// TIA Portal V17 export
// export: Created 2023-02-14T02:49:06.1157461Z, ExportSetting WithDefaults, DisplayName Totally Integrated Automation Portal, DisplayVersion V17, DisplayName TIA Portal Openness, DisplayVersion V17, DisplayName TIA Portal Teamcenter Gateway, DisplayVersion V17, DisplayName TIA Portal Version Control Interface, DisplayVersion V17, DisplayName SINAMICS Startdrive Advanced, DisplayVersion V17, DisplayName SINAMICS Startdrive G130, G150, S120, S150, SINAMICS MV, S210, DisplayVersion V17, DisplayName SINAMICS Startdrive G110M, G120, G120C, G120D, G120P, G115D, DisplayVersion V17, DisplayName STEP 7 Professional, DisplayVersion V17, DisplayName STEP 7 Safety, DisplayVersion V17, DisplayName WinCC Professional, DisplayVersion V17
FUNCTION_BLOCK "DOSE"   // FB102, LAD
TITLE = Dosing Module type 1; 1 adustable speed pump and 1 auto valve.
{ S7_Optimized_Access := 'FALSE' }
AUTHOR : N@wi
FAMILY : DOSE
NAME : DOSE
VERSION : 0.1
// Dosing Module type 1:
// Use for Dosing module with adjustable speed pump and auto valve. Coarse dosing 
// and Fine dosing by adjusting the pump speed.
// stored: AutoNumber false, IsIECCheckEnabled false, SetENOAutomatically false, UDAEnableTagReadback false
   VAR_INPUT
      ISTART_COND : Bool;   // Starting Condition. 1 = Dose sequence can be Start
      IOP_COND : Bool;   // Operating Condition. 0 = Dose will be hold
      V_CLOSE : Bool;   // Valve in close position
      V_OPEN : Bool;   // Valve in open position
      P_RUN : Bool;   // Pump Run
      P_STOP : Bool;   // Pump Stop
      OP_MODE : Bool := TRUE;   // Dosing Mode; 0 = MANUAL; 1 = AUTO
      ISTART_AUT : Bool;   // Start command in Auto dosing mode
      IHOLD_AUT : Bool;   // Hold command in Auto dosing mode
      ISTOP_AUT : Bool;   // Stop command in Auto dosing mode
      ICOMP_AUT : Bool;   // Complete command in Auto dosing mode
      MON_EN : Bool;   // Monitoring time enable
      "Pulse 1HZ" : Bool;
      ACT_QTY : Real;   // Actual Counter quantity
      MON_TIME : Real := 60.0;   // Monitoring Time (in second)
      SP_DOSEQTY : Real;   // Dosing Setpoint Quantity
      SP_FINEQTY : Real;   // Fine Quantity Setpoint
      SP_IdleSPEED : Real;
      SP_FINESPEED : Real;   // Fine Speed Setpoint
      SP_COARSESPEED : Real;   // Coarse Speed Setpoint
      SAMPLE_T : Real := 1.0;   // Sample Time
      SETTLE_T : Real := 3.0;   // Settling Time
      INF_PERC : Real := 2.0;   // Percentage of calculated infligh qty (in %)
      LDT : Date_And_Time;
   END_VAR
   VAR_OUTPUT
      QAUTO : Bool;   // Selected Operation Mode 0 = MANUAL; 1 = AUTO
      QIDLE : Bool;   // Dosing module in IDLE state
      QDOSERun : Bool;   // Dosing module in Running state
      QFinish : Bool;   // Dosing module in Finish
      QSTARTING : Bool;   // Dosing module in STARTING state
      QHOLDING : Bool;   // Dosing module in HOLDING state
      QHELD : Bool;   // Dosing module in HELD state
      QSTOPPING : Bool;   // Dosing module in STOPPING state
      QSTOPPED : Bool;   // Dosing module in STOPPED state
      QSTART_COND : Bool;   // Starting Condition are met
      QOP_COND : Bool;   // Operating Condition are met
      QERR : Bool;   // General Error
      QERR_MON : Bool;   // Error cause by runtime monitoring error
      QERR_OP : Bool;   // Error cause by operating condition not OK
      QERR_START : Bool;   // Error cause by start condition not OK
      P_CMD : Bool;   // Pump Start command
      V_CMD : Bool;   // Valve Open command
      COUNT_RESET : Bool;   // Counter reset command
      QDoseComplete : Bool;
      P_SPEED : Real;   // Pump speed setpoint
      DOSED_QTY : Real;   // Dosed quantity
      ACT_MON_TIME : Real;   // Actual Monitoring Time
      Dose_State : Word;
   END_VAR
   VAR_IN_OUT
      IQOPSTART : Bool;   // Start command by operator in Manual dosing mode
      IQOPHOLD : Bool;   // Hold command by operator in Manual dosing mode
      IQOPSTOP : Bool;   // Stop command by operator in Manual dosing mode
      IQOPCOMPLETE : Bool;   // Complete command by operator in Manual dosing mode
      IQRESET : Bool;   // Reset Error
      IQINFL_QTY : Real := 3.0e+0;   // Inflight quantity. Will be calculated in end of dosing for the next dosing.
      IQSTEP : Int;   // Actual step
      IQRB_STEP : Int;   // Roll Back Step
   END_VAR
   VAR DB_SPECIFIC
      b_IDLE : Bool;   // Dosing module in IDLE state
      b_Finish : Bool;   // Dosing module in Finish state
      b_STARTING : Bool;   // Dosing module in STARTING state
      b_HOLDING : Bool;   // Dosing module in HOLDING state
      b_HELD : Bool;   // Dosing module in HELD state
      b_STOPPING : Bool;   // Dosing module in STOPPING state
      b_STOPPED : Bool;   // Dosing module in STOPPED state
      b_START : Bool;   // Start command
      b_HOLD : Bool;   // Hold command
      b_STOP : Bool;   // Stop command
      b_COMP : Bool;   // Complete command
      b_START_AP : Bool;   // Start command Auto Pulse
      b_HOLD_AP : Bool;   // Hold command Auto Pulse
      b_STOP_AP : Bool;   // Stop command Auto Pulse
      b_COMP_AP : Bool;   // Complete command Auto Pulse
      b_START_MP : Bool;   // Start command Manual Pulse
      b_HOLD_MP : Bool;   // Hold command Manual Pulse
      b_STOP_MP : Bool;   // Stop command Manual Pulse
      b_COMP_MP : Bool;   // Complete command Manual Pulse
      b_ERR_MON : Bool;   // Error cause by runtime monitoring error
      b_ERR_OP : Bool;   // Error cause by operating condition not OK
      b_ERR_START : Bool;   // Error cause by start condition not OK
      PE_Setle : Bool;
      PE_Mon : Bool;
      CMD_STEP : Int;   // STEP command
      r_MON : Real;   // Actual Monitoring Time
      r_STOP : Real;   // Quantity to stop dosing
      r_FINE : Real;   // Quantity change to fine dosing
      r_SETTLE_T : Real;   // Settling Time
      r_INFLIGHT : Real;   // Saved inflight qty
      r_DIFF : Real;   // Dosed Qty - SP Quantity
      r_INFDIFF : Real;   // Diff of Inflight qty to be added to new inflight
      r_INFPERC { ExternalAccessible := 'False'; ExternalVisible := 'False'; ExternalWritable := 'False'} : Real;
      LDT_Start { S7_SetPoint := 'True'} : Date_And_Time;
      LDT_Finish : Date_And_Time;
      TimeDose : Time;
      LastTimeDose : Time;
      PE_LDTStart : Bool;
      PE_LDTFinish : Bool;
      PE_LDTStore : Bool;
      PE_QtyStart : Bool;
      PE_QtyFinish : Bool;
      PE_QtyStore : Bool;
      AlwaysON : Bool;
      LastQtyDose : Real;
   END_VAR
   VAR_TEMP   // added for the SCL form of the ladder/FBD networks
      _w1 : Bool;
      _w2 : Bool;
      _w3 : Bool;
      _w4 : Bool;
   END_VAR
BEGIN

REGION Network 1: AlwaysON
   // Copying the command step number to actual step number to avoid double step in 
   // one scan.
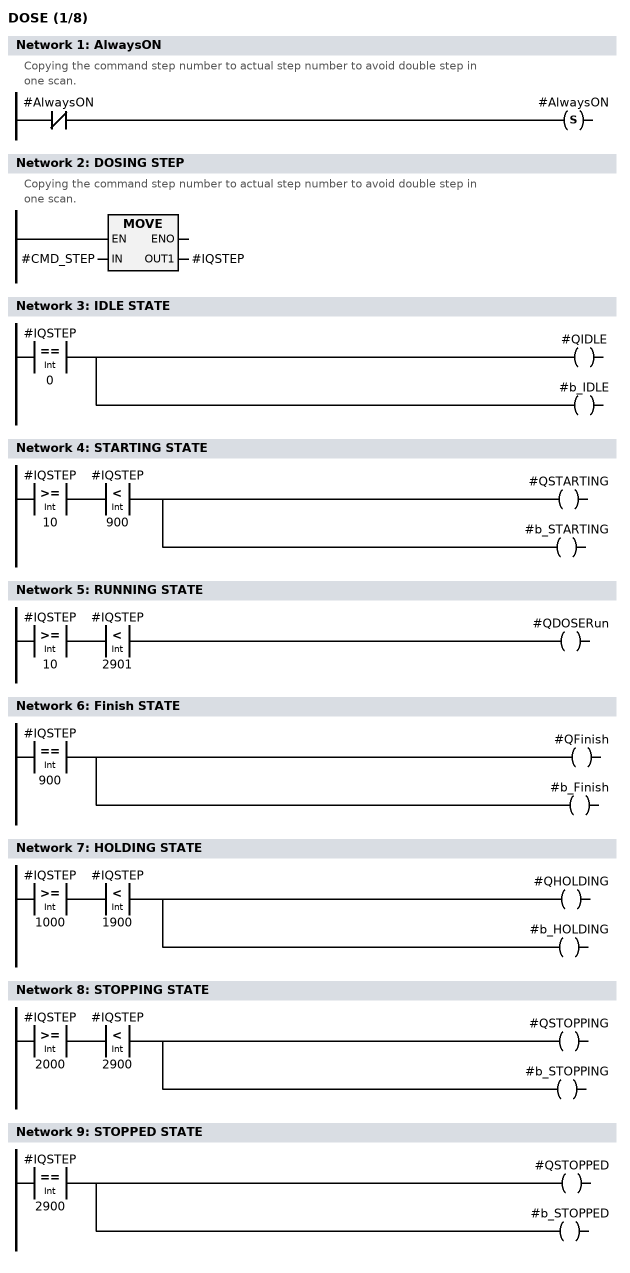
   RUNG wire#powerrail
      I_Contact( #AlwaysON )
      S_Coil( #AlwaysON )
   END_RUNG
   // the same network as SCL:
   IF NOT #AlwaysON THEN #AlwaysON := TRUE; END_IF;
END_REGION

REGION Network 2: DOSING STEP
   // Copying the command step number to actual step number to avoid double step in 
   // one scan.
   RUNG wire#powerrail
      { S7_GenerateENO := "TRUE" } Move(in := #CMD_STEP, out1 => #IQSTEP)
   END_RUNG
   // the same network as SCL:
   #IQSTEP := #CMD_STEP;
END_REGION

REGION Network 3: IDLE STATE
   RUNG wire#powerrail
      { S7_Templates := "SrcType := Int" } EQ_Contact(in1 := #IQSTEP, in2 := 0)
      wire#w1
      Coil( #QIDLE )
   END_RUNG
   RUNG wire#w1
      Coil( #b_IDLE )
   END_RUNG
   // the same network as SCL:
   #QIDLE := #IQSTEP = 0;
   #b_IDLE := #QIDLE;
END_REGION

REGION Network 4: STARTING STATE
   RUNG wire#powerrail
      { S7_Templates := "SrcType := Int" } GE_Contact(in1 := #IQSTEP, in2 := 10)
      { S7_Templates := "SrcType := Int" } LT_Contact(in1 := #IQSTEP, in2 := 900)
      wire#w1
      Coil( #QSTARTING )
   END_RUNG
   RUNG wire#w1
      Coil( #b_STARTING )
   END_RUNG
   // the same network as SCL:
   #QSTARTING := (#IQSTEP >= 10) AND (#IQSTEP < 900);
   #b_STARTING := #QSTARTING;
END_REGION

REGION Network 5: RUNNING STATE
   RUNG wire#powerrail
      { S7_Templates := "SrcType := Int" } GE_Contact(in1 := #IQSTEP, in2 := 10)
      { S7_Templates := "SrcType := Int" } LT_Contact(in1 := #IQSTEP, in2 := 2901)
      Coil( #QDOSERun )
   END_RUNG
   // the same network as SCL:
   #QDOSERun := (#IQSTEP >= 10) AND (#IQSTEP < 2901);
END_REGION

REGION Network 6: Finish STATE
   RUNG wire#powerrail
      { S7_Templates := "SrcType := Int" } EQ_Contact(in1 := #IQSTEP, in2 := 900)
      wire#w1
      Coil( #QFinish )
   END_RUNG
   RUNG wire#w1
      Coil( #b_Finish )
   END_RUNG
   // the same network as SCL:
   #QFinish := #IQSTEP = 900;
   #b_Finish := #QFinish;
END_REGION

REGION Network 7: HOLDING STATE
   RUNG wire#powerrail
      { S7_Templates := "SrcType := Int" } GE_Contact(in1 := #IQSTEP, in2 := 1000)
      { S7_Templates := "SrcType := Int" } LT_Contact(in1 := #IQSTEP, in2 := 1900)
      wire#w1
      Coil( #QHOLDING )
   END_RUNG
   RUNG wire#w1
      Coil( #b_HOLDING )
   END_RUNG
   // the same network as SCL:
   #QHOLDING := (#IQSTEP >= 1000) AND (#IQSTEP < 1900);
   #b_HOLDING := #QHOLDING;
END_REGION

REGION Network 8: STOPPING STATE
   RUNG wire#powerrail
      { S7_Templates := "SrcType := Int" } GE_Contact(in1 := #IQSTEP, in2 := 2000)
      { S7_Templates := "SrcType := Int" } LT_Contact(in1 := #IQSTEP, in2 := 2900)
      wire#w1
      Coil( #QSTOPPING )
   END_RUNG
   RUNG wire#w1
      Coil( #b_STOPPING )
   END_RUNG
   // the same network as SCL:
   #QSTOPPING := (#IQSTEP >= 2000) AND (#IQSTEP < 2900);
   #b_STOPPING := #QSTOPPING;
END_REGION

REGION Network 9: STOPPED STATE
   RUNG wire#powerrail
      { S7_Templates := "SrcType := Int" } EQ_Contact(in1 := #IQSTEP, in2 := 2900)
      wire#w1
      Coil( #QSTOPPED )
   END_RUNG
   RUNG wire#w1
      Coil( #b_STOPPED )
   END_RUNG
   // the same network as SCL:
   #QSTOPPED := #IQSTEP = 2900;
   #b_STOPPED := #QSTOPPED;
END_REGION

REGION Network 10: START COMMAND
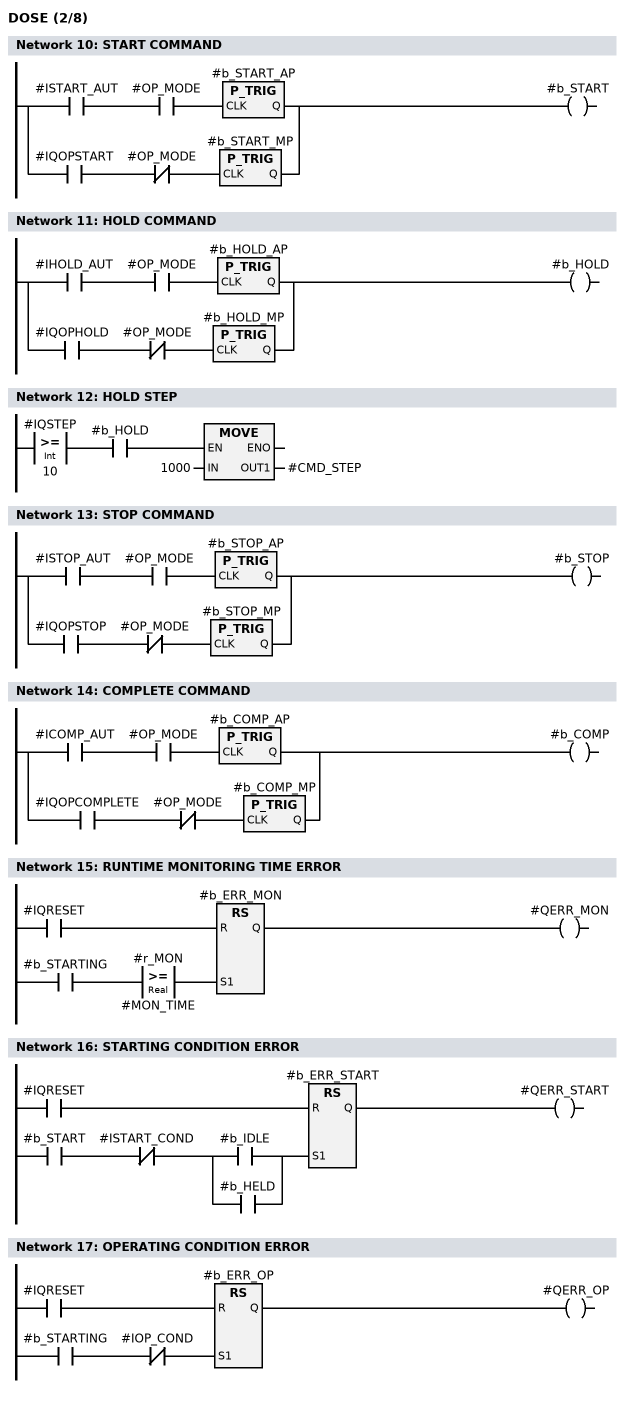
   RUNG wire#powerrail
      Contact( #ISTART_AUT )
      Contact( #OP_MODE )
      P_Trig( #b_START_AP )
      wire#w1
      Coil( #b_START )
   END_RUNG
   RUNG wire#powerrail
      Contact( #IQOPSTART )
      I_Contact( #OP_MODE )
      P_Trig( #b_START_MP )
   END_RUNG wire#w1
   // the same network as SCL:
   #_w1 := #ISTART_AUT AND #OP_MODE;
   #_w2 := #_w1 AND NOT #b_START_AP;   // rising edge
   #b_START_AP := #_w1;
   #_w3 := #IQOPSTART AND NOT #OP_MODE;
   #_w4 := #_w3 AND NOT #b_START_MP;   // rising edge
   #b_START_MP := #_w3;
   #b_START := #_w2 OR #_w4;
END_REGION

REGION Network 11: HOLD COMMAND
   RUNG wire#powerrail
      Contact( #IHOLD_AUT )
      Contact( #OP_MODE )
      P_Trig( #b_HOLD_AP )
      wire#w1
      Coil( #b_HOLD )
   END_RUNG
   RUNG wire#powerrail
      Contact( #IQOPHOLD )
      I_Contact( #OP_MODE )
      P_Trig( #b_HOLD_MP )
   END_RUNG wire#w1
   // the same network as SCL:
   #_w1 := #IHOLD_AUT AND #OP_MODE;
   #_w2 := #_w1 AND NOT #b_HOLD_AP;   // rising edge
   #b_HOLD_AP := #_w1;
   #_w3 := #IQOPHOLD AND NOT #OP_MODE;
   #_w4 := #_w3 AND NOT #b_HOLD_MP;   // rising edge
   #b_HOLD_MP := #_w3;
   #b_HOLD := #_w2 OR #_w4;
END_REGION

REGION Network 12: HOLD STEP
   RUNG wire#powerrail
      { S7_Templates := "SrcType := Int" } GE_Contact(in1 := #IQSTEP, in2 := 10)
      Contact( #b_HOLD )
      { S7_GenerateENO := "TRUE" } Move(in := 1000, out1 => #CMD_STEP)
   END_RUNG
   // the same network as SCL:
   IF (#IQSTEP >= 10) AND #b_HOLD THEN #CMD_STEP := 1000; END_IF;
END_REGION

REGION Network 13: STOP COMMAND
   RUNG wire#powerrail
      Contact( #ISTOP_AUT )
      Contact( #OP_MODE )
      P_Trig( #b_STOP_AP )
      wire#w1
      Coil( #b_STOP )
   END_RUNG
   RUNG wire#powerrail
      Contact( #IQOPSTOP )
      I_Contact( #OP_MODE )
      P_Trig( #b_STOP_MP )
   END_RUNG wire#w1
   // the same network as SCL:
   #_w1 := #ISTOP_AUT AND #OP_MODE;
   #_w2 := #_w1 AND NOT #b_STOP_AP;   // rising edge
   #b_STOP_AP := #_w1;
   #_w3 := #IQOPSTOP AND NOT #OP_MODE;
   #_w4 := #_w3 AND NOT #b_STOP_MP;   // rising edge
   #b_STOP_MP := #_w3;
   #b_STOP := #_w2 OR #_w4;
END_REGION

REGION Network 14: COMPLETE COMMAND
   RUNG wire#powerrail
      Contact( #ICOMP_AUT )
      Contact( #OP_MODE )
      P_Trig( #b_COMP_AP )
      wire#w1
      Coil( #b_COMP )
   END_RUNG
   RUNG wire#powerrail
      Contact( #IQOPCOMPLETE )
      I_Contact( #OP_MODE )
      P_Trig( #b_COMP_MP )
   END_RUNG wire#w1
   // the same network as SCL:
   #_w1 := #ICOMP_AUT AND #OP_MODE;
   #_w2 := #_w1 AND NOT #b_COMP_AP;   // rising edge
   #b_COMP_AP := #_w1;
   #_w3 := #IQOPCOMPLETE AND NOT #OP_MODE;
   #_w4 := #_w3 AND NOT #b_COMP_MP;   // rising edge
   #b_COMP_MP := #_w3;
   #b_COMP := #_w2 OR #_w4;
END_REGION

REGION Network 15: RUNTIME MONITORING TIME ERROR
   RUNG wire#powerrail
      Contact( #IQRESET )
      S_RS(operand := #b_ERR_MON, s1 := wire#w1)
      Coil( #QERR_MON )
   END_RUNG
   RUNG wire#powerrail
      Contact( #b_STARTING )
      { S7_Templates := "SrcType := Real" } GE_Contact(in1 := #r_MON, in2 := #MON_TIME)
   END_RUNG wire#w1
   // the same network as SCL:
   IF #IQRESET THEN
       #b_ERR_MON := FALSE;   // RS flip-flop
   END_IF;
   IF #b_STARTING AND (#r_MON >= #MON_TIME) THEN #b_ERR_MON := TRUE; END_IF;
   #QERR_MON := #b_ERR_MON;
END_REGION

REGION Network 16: STARTING CONDITION ERROR
   RUNG wire#powerrail
      Contact( #IQRESET )
      S_RS(operand := #b_ERR_START, s1 := wire#w2)
      Coil( #QERR_START )
   END_RUNG
   RUNG wire#powerrail
      Contact( #b_START )
      I_Contact( #ISTART_COND )
      wire#w1
      Contact( #b_IDLE )
   END_RUNG wire#w2
   RUNG wire#w1
      Contact( #b_HELD )
   END_RUNG wire#w2
   // the same network as SCL:
   IF #IQRESET THEN
       #b_ERR_START := FALSE;   // RS flip-flop
   END_IF;
   IF #b_START AND NOT #ISTART_COND AND (#b_IDLE OR #b_HELD) THEN #b_ERR_START := TRUE; END_IF;
   #QERR_START := #b_ERR_START;
END_REGION

REGION Network 17: OPERATING CONDITION ERROR
   RUNG wire#powerrail
      Contact( #IQRESET )
      S_RS(operand := #b_ERR_OP, s1 := wire#w1)
      Coil( #QERR_OP )
   END_RUNG
   RUNG wire#powerrail
      Contact( #b_STARTING )
      I_Contact( #IOP_COND )
   END_RUNG wire#w1
   // the same network as SCL:
   IF #IQRESET THEN
       #b_ERR_OP := FALSE;   // RS flip-flop
   END_IF;
   IF #b_STARTING AND NOT #IOP_COND THEN #b_ERR_OP := TRUE; END_IF;
   #QERR_OP := #b_ERR_OP;
END_REGION

REGION Network 18: GENERAL ERROR
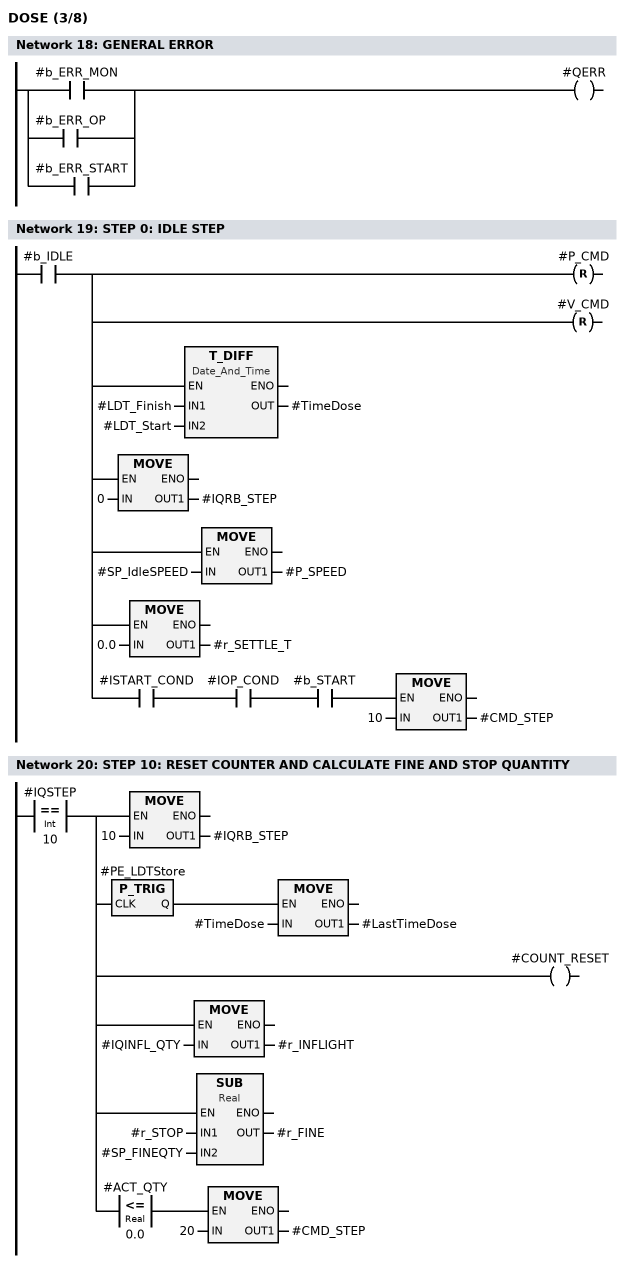
   RUNG wire#powerrail
      Contact( #b_ERR_MON )
      wire#w1
      Coil( #QERR )
   END_RUNG
   RUNG wire#powerrail
      Contact( #b_ERR_OP )
   END_RUNG wire#w1
   RUNG wire#powerrail
      Contact( #b_ERR_START )
   END_RUNG wire#w1
   // the same network as SCL:
   #QERR := #b_ERR_MON OR #b_ERR_OP OR #b_ERR_START;
END_REGION

REGION Network 19: STEP 0: IDLE STEP
   RUNG wire#powerrail
      Contact( #b_IDLE )
      wire#w1
      R_Coil( #P_CMD )
   END_RUNG
   RUNG wire#w1
      R_Coil( #V_CMD )
   END_RUNG
   RUNG wire#w1
      { S7_Templates := "[date_type := Date_And_Time, time_type := Time]" } T_DIFF(IN1 := #LDT_Finish, IN2 := #LDT_Start, OUT => #TimeDose)
   END_RUNG
   RUNG wire#w1
      { S7_GenerateENO := "TRUE" } Move(in := 0, out1 => #IQRB_STEP)
   END_RUNG
   RUNG wire#w1
      { S7_GenerateENO := "TRUE" } Move(in := #SP_IdleSPEED, out1 => #P_SPEED)
   END_RUNG
   RUNG wire#w1
      { S7_GenerateENO := "TRUE" } Move(in := 0.0, out1 => #r_SETTLE_T)
   END_RUNG
   RUNG wire#w1
      Contact( #ISTART_COND )
      Contact( #IOP_COND )
      Contact( #b_START )
      { S7_GenerateENO := "TRUE" } Move(in := 10, out1 => #CMD_STEP)
   END_RUNG
   // the same network as SCL:
   IF #b_IDLE THEN
       #P_CMD := FALSE;
       #V_CMD := FALSE;
       T_DIFF(IN1 := #LDT_Finish, IN2 := #LDT_Start, OUT => #TimeDose);
       #IQRB_STEP := 0;
       #P_SPEED := #SP_IdleSPEED;
       #r_SETTLE_T := 0.0;
   END_IF;
   IF #b_IDLE AND #ISTART_COND AND #IOP_COND AND #b_START THEN #CMD_STEP := 10; END_IF;
END_REGION

REGION Network 20: STEP 10: RESET COUNTER AND CALCULATE FINE AND STOP QUANTITY
   RUNG wire#powerrail
      { S7_Templates := "SrcType := Int" } EQ_Contact(in1 := #IQSTEP, in2 := 10)
      wire#w1
      { S7_GenerateENO := "TRUE" } Move(in := 10, out1 => #IQRB_STEP)
   END_RUNG
   RUNG wire#w1
      P_Trig( #PE_LDTStore )
      Move(in := #TimeDose, out1 => #LastTimeDose)
   END_RUNG
   RUNG wire#w1
      Coil( #COUNT_RESET )
   END_RUNG
   RUNG wire#w1
      { S7_GenerateENO := "TRUE" } Move(in := #IQINFL_QTY, out1 => #r_INFLIGHT)
   END_RUNG
   RUNG wire#w1
      { S7_Templates := "SrcType := Real"; S7_GenerateENO := "TRUE" } Sub(in1 := #r_STOP, in2 := #SP_FINEQTY, out => #r_FINE)
   END_RUNG
   RUNG wire#w1
      { S7_Templates := "SrcType := Real" } LE_Contact(in1 := #ACT_QTY, in2 := 0.0)
      { S7_GenerateENO := "TRUE" } Move(in := 20, out1 => #CMD_STEP)
   END_RUNG
   // the same network as SCL:
   #_w1 := #IQSTEP = 10;
   IF #_w1 THEN #IQRB_STEP := 10; END_IF;
   #_w2 := #_w1 AND NOT #PE_LDTStore;   // rising edge
   #PE_LDTStore := #_w1;
   IF #_w2 THEN #LastTimeDose := #TimeDose; END_IF;
   #COUNT_RESET := #_w1;
   IF #_w1 THEN
       #r_INFLIGHT := #IQINFL_QTY;
       #r_FINE := #r_STOP - #SP_FINEQTY;
   END_IF;
   IF #_w1 AND (#ACT_QTY <= 0.0) THEN #CMD_STEP := 20; END_IF;
END_REGION

REGION Network 21: STEP 20: OPEN VALVE
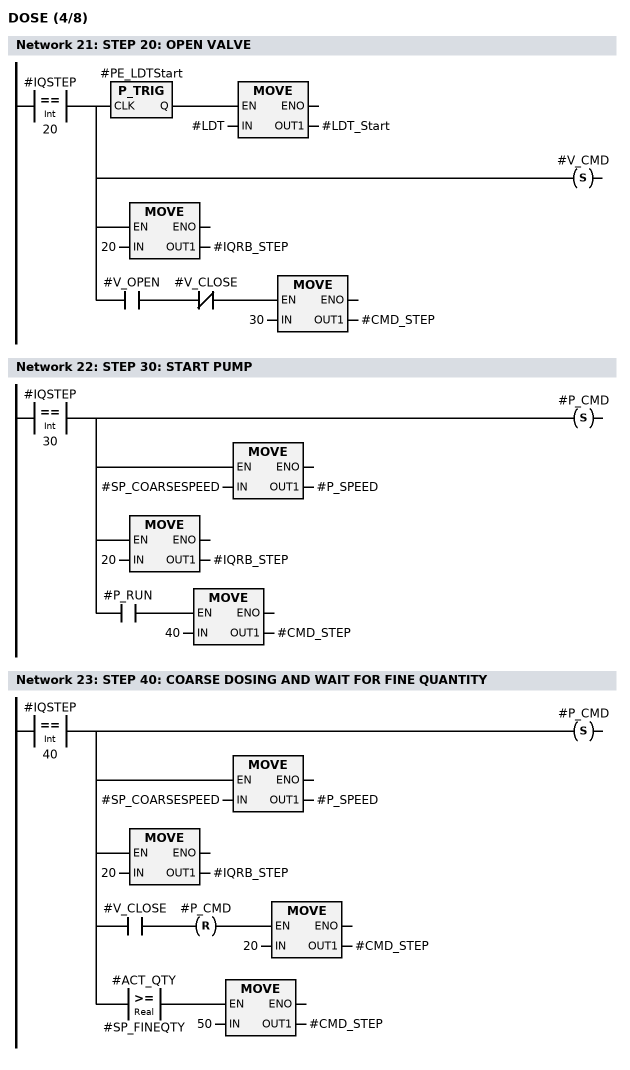
   RUNG wire#powerrail
      { S7_Templates := "SrcType := Int" } EQ_Contact(in1 := #IQSTEP, in2 := 20)
      wire#w1
      P_Trig( #PE_LDTStart )
      Move(in := #LDT, out1 => #LDT_Start)
   END_RUNG
   RUNG wire#w1
      S_Coil( #V_CMD )
   END_RUNG
   RUNG wire#w1
      { S7_GenerateENO := "TRUE" } Move(in := 20, out1 => #IQRB_STEP)
   END_RUNG
   RUNG wire#w1
      Contact( #V_OPEN )
      I_Contact( #V_CLOSE )
      { S7_GenerateENO := "TRUE" } Move(in := 30, out1 => #CMD_STEP)
   END_RUNG
   // the same network as SCL:
   #_w1 := #IQSTEP = 20;
   #_w2 := #_w1 AND NOT #PE_LDTStart;   // rising edge
   #PE_LDTStart := #_w1;
   IF #_w2 THEN #LDT_Start := #LDT; END_IF;
   IF #_w1 THEN
       #V_CMD := TRUE;
       #IQRB_STEP := 20;
   END_IF;
   IF #_w1 AND #V_OPEN AND NOT #V_CLOSE THEN #CMD_STEP := 30; END_IF;
END_REGION

REGION Network 22: STEP 30: START PUMP
   RUNG wire#powerrail
      { S7_Templates := "SrcType := Int" } EQ_Contact(in1 := #IQSTEP, in2 := 30)
      wire#w1
      S_Coil( #P_CMD )
   END_RUNG
   RUNG wire#w1
      { S7_GenerateENO := "TRUE" } Move(in := #SP_COARSESPEED, out1 => #P_SPEED)
   END_RUNG
   RUNG wire#w1
      { S7_GenerateENO := "TRUE" } Move(in := 20, out1 => #IQRB_STEP)
   END_RUNG
   RUNG wire#w1
      Contact( #P_RUN )
      { S7_GenerateENO := "TRUE" } Move(in := 40, out1 => #CMD_STEP)
   END_RUNG
   // the same network as SCL:
   #_w1 := #IQSTEP = 30;
   IF #_w1 THEN
       #P_CMD := TRUE;
       #P_SPEED := #SP_COARSESPEED;
       #IQRB_STEP := 20;
   END_IF;
   IF #_w1 AND #P_RUN THEN #CMD_STEP := 40; END_IF;
END_REGION

REGION Network 23: STEP 40: COARSE DOSING AND WAIT FOR FINE QUANTITY
   RUNG wire#powerrail
      { S7_Templates := "SrcType := Int" } EQ_Contact(in1 := #IQSTEP, in2 := 40)
      wire#w1
      S_Coil( #P_CMD )
   END_RUNG
   RUNG wire#w1
      { S7_GenerateENO := "TRUE" } Move(in := #SP_COARSESPEED, out1 => #P_SPEED)
   END_RUNG
   RUNG wire#w1
      { S7_GenerateENO := "TRUE" } Move(in := 20, out1 => #IQRB_STEP)
   END_RUNG
   RUNG wire#w1
      Contact( #V_CLOSE )
      R_Coil( #P_CMD )
      { S7_GenerateENO := "TRUE" } Move(in := 20, out1 => #CMD_STEP)
   END_RUNG
   RUNG wire#w1
      { S7_Templates := "SrcType := Real" } GE_Contact(in1 := #ACT_QTY, in2 := #SP_FINEQTY)
      { S7_GenerateENO := "TRUE" } Move(in := 50, out1 => #CMD_STEP)
   END_RUNG
   // the same network as SCL:
   #_w1 := #IQSTEP = 40;
   IF #_w1 THEN
       #P_CMD := TRUE;
       #P_SPEED := #SP_COARSESPEED;
       #IQRB_STEP := 20;
   END_IF;
   IF #_w1 AND #V_CLOSE THEN
       #P_CMD := FALSE;
       #CMD_STEP := 20;
   END_IF;
   IF #_w1 AND (#ACT_QTY >= #SP_FINEQTY) THEN #CMD_STEP := 50; END_IF;
END_REGION

REGION Network 24: STEP 50: FINE DOSING AND WAIT FOR STOP QUANTITY
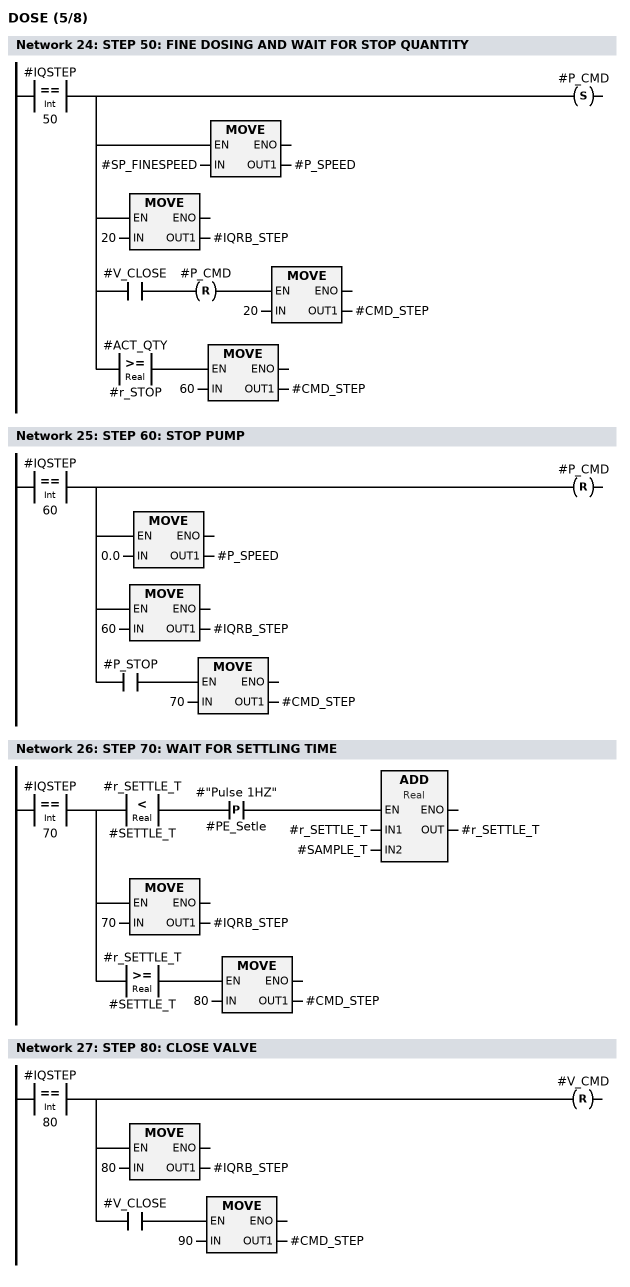
   RUNG wire#powerrail
      { S7_Templates := "SrcType := Int" } EQ_Contact(in1 := #IQSTEP, in2 := 50)
      wire#w1
      S_Coil( #P_CMD )
   END_RUNG
   RUNG wire#w1
      { S7_GenerateENO := "TRUE" } Move(in := #SP_FINESPEED, out1 => #P_SPEED)
   END_RUNG
   RUNG wire#w1
      { S7_GenerateENO := "TRUE" } Move(in := 20, out1 => #IQRB_STEP)
   END_RUNG
   RUNG wire#w1
      Contact( #V_CLOSE )
      R_Coil( #P_CMD )
      { S7_GenerateENO := "TRUE" } Move(in := 20, out1 => #CMD_STEP)
   END_RUNG
   RUNG wire#w1
      { S7_Templates := "SrcType := Real" } GE_Contact(in1 := #ACT_QTY, in2 := #r_STOP)
      { S7_GenerateENO := "TRUE" } Move(in := 60, out1 => #CMD_STEP)
   END_RUNG
   // the same network as SCL:
   #_w1 := #IQSTEP = 50;
   IF #_w1 THEN
       #P_CMD := TRUE;
       #P_SPEED := #SP_FINESPEED;
       #IQRB_STEP := 20;
   END_IF;
   IF #_w1 AND #V_CLOSE THEN
       #P_CMD := FALSE;
       #CMD_STEP := 20;
   END_IF;
   IF #_w1 AND (#ACT_QTY >= #r_STOP) THEN #CMD_STEP := 60; END_IF;
END_REGION

REGION Network 25: STEP 60: STOP PUMP
   RUNG wire#powerrail
      { S7_Templates := "SrcType := Int" } EQ_Contact(in1 := #IQSTEP, in2 := 60)
      wire#w1
      R_Coil( #P_CMD )
   END_RUNG
   RUNG wire#w1
      { S7_GenerateENO := "TRUE" } Move(in := 0.0, out1 => #P_SPEED)
   END_RUNG
   RUNG wire#w1
      { S7_GenerateENO := "TRUE" } Move(in := 60, out1 => #IQRB_STEP)
   END_RUNG
   RUNG wire#w1
      Contact( #P_STOP )
      { S7_GenerateENO := "TRUE" } Move(in := 70, out1 => #CMD_STEP)
   END_RUNG
   // the same network as SCL:
   #_w1 := #IQSTEP = 60;
   IF #_w1 THEN
       #P_CMD := FALSE;
       #P_SPEED := 0.0;
       #IQRB_STEP := 60;
   END_IF;
   IF #_w1 AND #P_STOP THEN #CMD_STEP := 70; END_IF;
END_REGION

REGION Network 26: STEP 70: WAIT FOR SETTLING TIME
   RUNG wire#powerrail
      { S7_Templates := "SrcType := Int" } EQ_Contact(in1 := #IQSTEP, in2 := 70)
      wire#w1
      { S7_Templates := "SrcType := Real" } LT_Contact(in1 := #r_SETTLE_T, in2 := #SETTLE_T)
      P_Contact(operand := #"Pulse 1HZ", bit := #PE_Setle)
      { S7_Templates := "SrcType := Real"; S7_GenerateENO := "TRUE" } Add(in1 := #r_SETTLE_T, in2 := #SAMPLE_T, out => #r_SETTLE_T)
   END_RUNG
   RUNG wire#w1
      { S7_GenerateENO := "TRUE" } Move(in := 70, out1 => #IQRB_STEP)
   END_RUNG
   RUNG wire#w1
      { S7_Templates := "SrcType := Real" } GE_Contact(in1 := #r_SETTLE_T, in2 := #SETTLE_T)
      { S7_GenerateENO := "TRUE" } Move(in := 80, out1 => #CMD_STEP)
   END_RUNG
   // the same network as SCL:
   #_w1 := #IQSTEP = 70;
   #_w2 := #_w1 AND (#r_SETTLE_T < #SETTLE_T) AND #"Pulse 1HZ" AND NOT #PE_Setle;   // rising edge of #"Pulse 1HZ"
   #PE_Setle := #"Pulse 1HZ";
   IF #_w2 THEN #r_SETTLE_T := #r_SETTLE_T + #SAMPLE_T; END_IF;
   IF #_w1 THEN #IQRB_STEP := 70; END_IF;
   IF #_w1 AND (#r_SETTLE_T >= #SETTLE_T) THEN #CMD_STEP := 80; END_IF;
END_REGION

REGION Network 27: STEP 80: CLOSE VALVE
   RUNG wire#powerrail
      { S7_Templates := "SrcType := Int" } EQ_Contact(in1 := #IQSTEP, in2 := 80)
      wire#w1
      R_Coil( #V_CMD )
   END_RUNG
   RUNG wire#w1
      { S7_GenerateENO := "TRUE" } Move(in := 80, out1 => #IQRB_STEP)
   END_RUNG
   RUNG wire#w1
      Contact( #V_CLOSE )
      { S7_GenerateENO := "TRUE" } Move(in := 90, out1 => #CMD_STEP)
   END_RUNG
   // the same network as SCL:
   #_w1 := #IQSTEP = 80;
   IF #_w1 THEN
       #V_CMD := FALSE;
       #IQRB_STEP := 80;
   END_IF;
   IF #_w1 AND #V_CLOSE THEN #CMD_STEP := 90; END_IF;
END_REGION

REGION Network 28: STEP 90: CALCULATE INFLIGHT QTY
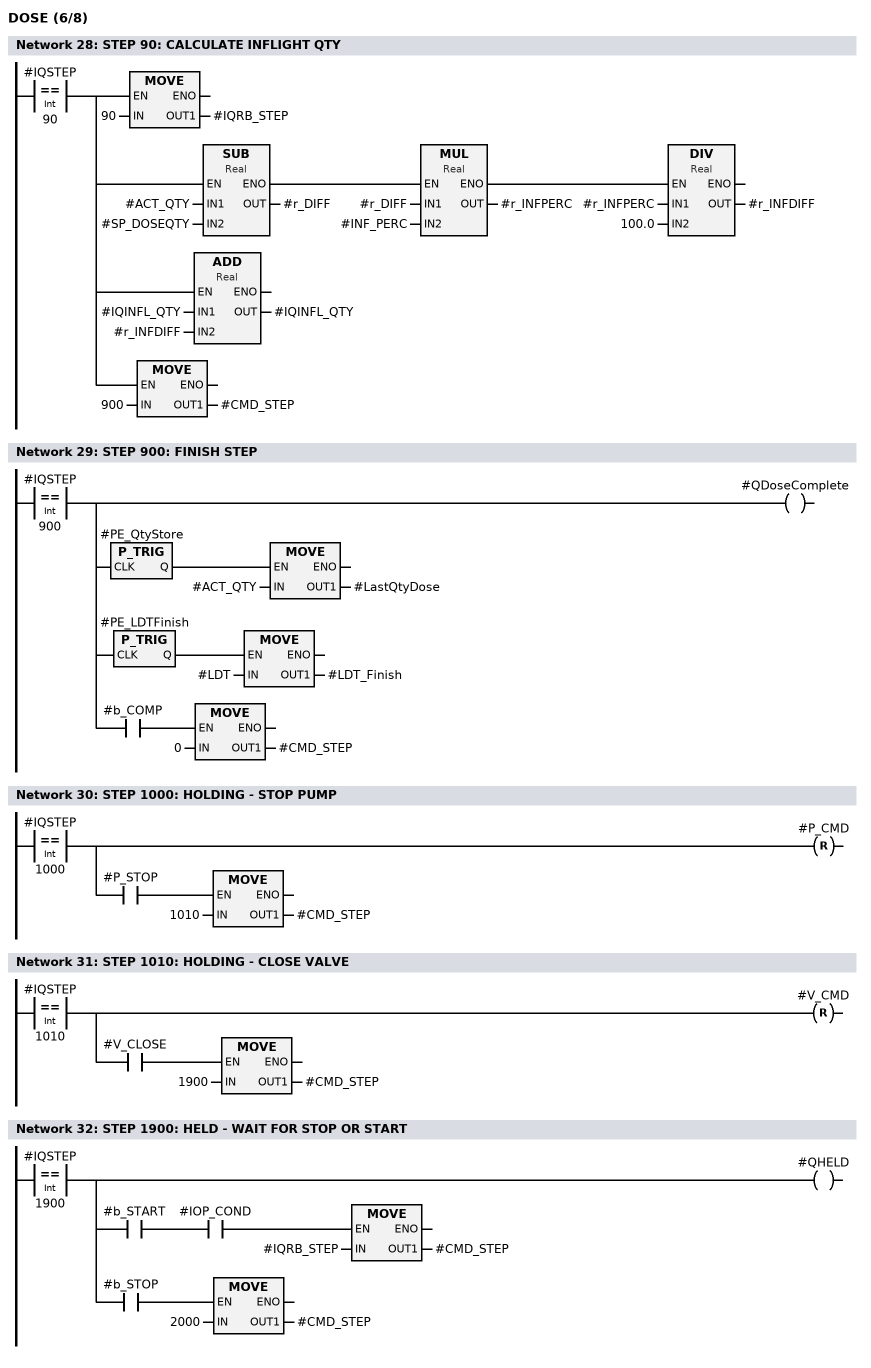
   RUNG wire#powerrail
      { S7_Templates := "SrcType := Int" } EQ_Contact(in1 := #IQSTEP, in2 := 90)
      wire#w1
      { S7_GenerateENO := "TRUE" } Move(in := 90, out1 => #IQRB_STEP)
   END_RUNG
   RUNG wire#w1
      { S7_Templates := "SrcType := Real"; S7_GenerateENO := "TRUE" } Sub(in1 := #ACT_QTY, in2 := #SP_DOSEQTY, out => #r_DIFF)
      { S7_Templates := "SrcType := Real"; S7_GenerateENO := "TRUE" } Mul(in1 := #r_DIFF, in2 := #INF_PERC, out => #r_INFPERC)
      { S7_Templates := "SrcType := Real"; S7_GenerateENO := "TRUE" } Div(in1 := #r_INFPERC, in2 := 100.0, out => #r_INFDIFF)
   END_RUNG
   RUNG wire#w1
      { S7_Templates := "SrcType := Real"; S7_GenerateENO := "TRUE" } Add(in1 := #IQINFL_QTY, in2 := #r_INFDIFF, out => #IQINFL_QTY)
   END_RUNG
   RUNG wire#w1
      { S7_GenerateENO := "TRUE" } Move(in := 900, out1 => #CMD_STEP)
   END_RUNG
   // the same network as SCL:
   // ENO of a box is taken as its EN; it also drops when the box reports an error
   IF #IQSTEP = 90 THEN
       #IQRB_STEP := 90;
       #r_DIFF := #ACT_QTY - #SP_DOSEQTY;
       #r_INFPERC := #r_DIFF * #INF_PERC;
       #r_INFDIFF := #r_INFPERC / 100.0;
       #IQINFL_QTY := #IQINFL_QTY + #r_INFDIFF;
       #CMD_STEP := 900;
   END_IF;
END_REGION

REGION Network 29: STEP 900: FINISH STEP
   RUNG wire#powerrail
      { S7_Templates := "SrcType := Int" } EQ_Contact(in1 := #IQSTEP, in2 := 900)
      wire#w1
      Coil( #QDoseComplete )
   END_RUNG
   RUNG wire#w1
      P_Trig( #PE_QtyStore )
      Move(in := #ACT_QTY, out1 => #LastQtyDose)
   END_RUNG
   RUNG wire#w1
      P_Trig( #PE_LDTFinish )
      Move(in := #LDT, out1 => #LDT_Finish)
   END_RUNG
   RUNG wire#w1
      Contact( #b_COMP )
      { S7_GenerateENO := "TRUE" } Move(in := 0, out1 => #CMD_STEP)
   END_RUNG
   // the same network as SCL:
   #QDoseComplete := #IQSTEP = 900;
   #_w1 := #QDoseComplete AND NOT #PE_QtyStore;   // rising edge
   #PE_QtyStore := #QDoseComplete;
   IF #_w1 THEN #LastQtyDose := #ACT_QTY; END_IF;
   #_w2 := #QDoseComplete AND NOT #PE_LDTFinish;   // rising edge
   #PE_LDTFinish := #QDoseComplete;
   IF #_w2 THEN #LDT_Finish := #LDT; END_IF;
   IF #QDoseComplete AND #b_COMP THEN #CMD_STEP := 0; END_IF;
END_REGION

REGION Network 30: STEP 1000: HOLDING - STOP PUMP
   RUNG wire#powerrail
      { S7_Templates := "SrcType := Int" } EQ_Contact(in1 := #IQSTEP, in2 := 1000)
      wire#w1
      R_Coil( #P_CMD )
   END_RUNG
   RUNG wire#w1
      Contact( #P_STOP )
      { S7_GenerateENO := "TRUE" } Move(in := 1010, out1 => #CMD_STEP)
   END_RUNG
   // the same network as SCL:
   #_w1 := #IQSTEP = 1000;
   IF #_w1 THEN #P_CMD := FALSE; END_IF;
   IF #_w1 AND #P_STOP THEN #CMD_STEP := 1010; END_IF;
END_REGION

REGION Network 31: STEP 1010: HOLDING - CLOSE VALVE
   RUNG wire#powerrail
      { S7_Templates := "SrcType := Int" } EQ_Contact(in1 := #IQSTEP, in2 := 1010)
      wire#w1
      R_Coil( #V_CMD )
   END_RUNG
   RUNG wire#w1
      Contact( #V_CLOSE )
      { S7_GenerateENO := "TRUE" } Move(in := 1900, out1 => #CMD_STEP)
   END_RUNG
   // the same network as SCL:
   #_w1 := #IQSTEP = 1010;
   IF #_w1 THEN #V_CMD := FALSE; END_IF;
   IF #_w1 AND #V_CLOSE THEN #CMD_STEP := 1900; END_IF;
END_REGION

REGION Network 32: STEP 1900: HELD - WAIT FOR STOP OR START
   RUNG wire#powerrail
      { S7_Templates := "SrcType := Int" } EQ_Contact(in1 := #IQSTEP, in2 := 1900)
      wire#w1
      Coil( #QHELD )
   END_RUNG
   RUNG wire#w1
      Contact( #b_START )
      Contact( #IOP_COND )
      { S7_GenerateENO := "TRUE" } Move(in := #IQRB_STEP, out1 => #CMD_STEP)
   END_RUNG
   RUNG wire#w1
      Contact( #b_STOP )
      { S7_GenerateENO := "TRUE" } Move(in := 2000, out1 => #CMD_STEP)
   END_RUNG
   // the same network as SCL:
   #QHELD := #IQSTEP = 1900;
   IF #QHELD AND #b_START AND #IOP_COND THEN #CMD_STEP := #IQRB_STEP; END_IF;
   IF #QHELD AND #b_STOP THEN #CMD_STEP := 2000; END_IF;
END_REGION

REGION Network 33: STEP 2000: STOPPING - STOP PUMP
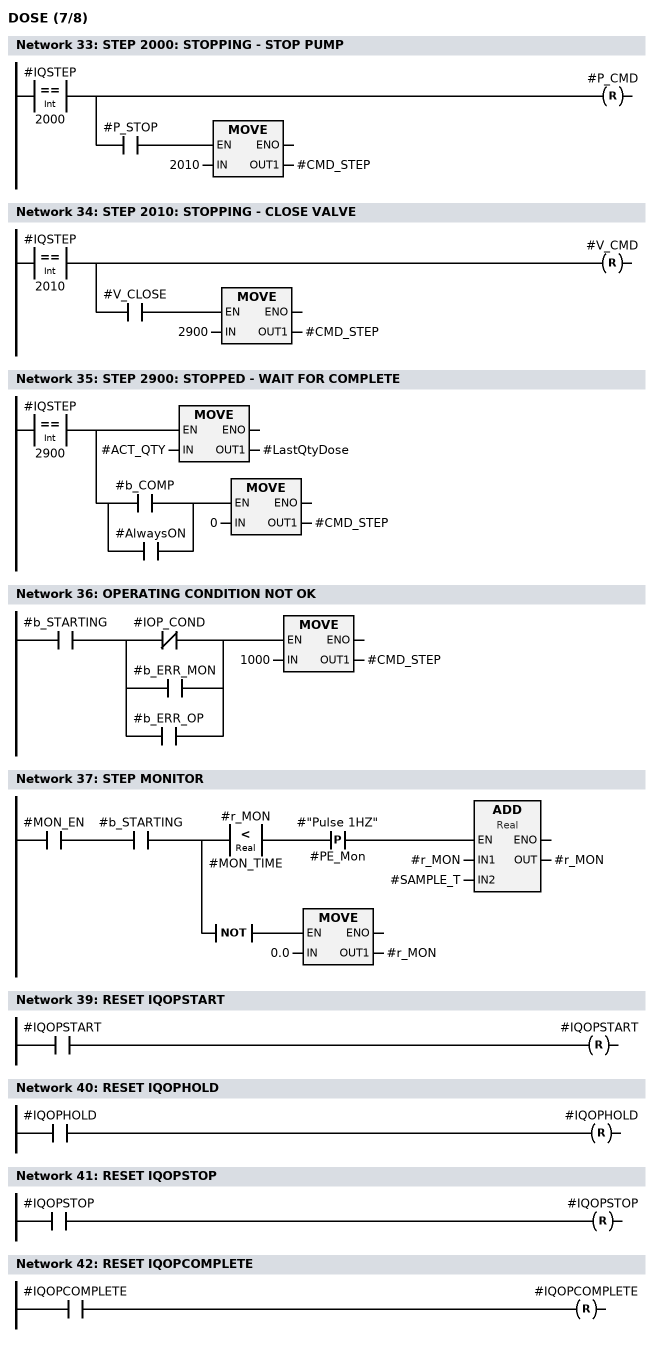
   RUNG wire#powerrail
      { S7_Templates := "SrcType := Int" } EQ_Contact(in1 := #IQSTEP, in2 := 2000)
      wire#w1
      R_Coil( #P_CMD )
   END_RUNG
   RUNG wire#w1
      Contact( #P_STOP )
      { S7_GenerateENO := "TRUE" } Move(in := 2010, out1 => #CMD_STEP)
   END_RUNG
   // the same network as SCL:
   #_w1 := #IQSTEP = 2000;
   IF #_w1 THEN #P_CMD := FALSE; END_IF;
   IF #_w1 AND #P_STOP THEN #CMD_STEP := 2010; END_IF;
END_REGION

REGION Network 34: STEP 2010: STOPPING - CLOSE VALVE
   RUNG wire#powerrail
      { S7_Templates := "SrcType := Int" } EQ_Contact(in1 := #IQSTEP, in2 := 2010)
      wire#w1
      R_Coil( #V_CMD )
   END_RUNG
   RUNG wire#w1
      Contact( #V_CLOSE )
      { S7_GenerateENO := "TRUE" } Move(in := 2900, out1 => #CMD_STEP)
   END_RUNG
   // the same network as SCL:
   #_w1 := #IQSTEP = 2010;
   IF #_w1 THEN #V_CMD := FALSE; END_IF;
   IF #_w1 AND #V_CLOSE THEN #CMD_STEP := 2900; END_IF;
END_REGION

REGION Network 35: STEP 2900: STOPPED - WAIT FOR COMPLETE
   RUNG wire#powerrail
      { S7_Templates := "SrcType := Int" } EQ_Contact(in1 := #IQSTEP, in2 := 2900)
      wire#w1
      Move(in := #ACT_QTY, out1 => #LastQtyDose)
   END_RUNG
   RUNG wire#w1
      Contact( #b_COMP )
      wire#w2
      { S7_GenerateENO := "TRUE" } Move(in := 0, out1 => #CMD_STEP)
   END_RUNG
   RUNG wire#w1
      Contact( #AlwaysON )
   END_RUNG wire#w2
   // the same network as SCL:
   #_w1 := #IQSTEP = 2900;
   IF #_w1 THEN #LastQtyDose := #ACT_QTY; END_IF;
   IF #_w1 AND (#b_COMP OR #AlwaysON) THEN #CMD_STEP := 0; END_IF;
END_REGION

REGION Network 36: OPERATING CONDITION NOT OK
   RUNG wire#powerrail
      Contact( #b_STARTING )
      wire#w1
      I_Contact( #IOP_COND )
      wire#w2
      { S7_GenerateENO := "TRUE" } Move(in := 1000, out1 => #CMD_STEP)
   END_RUNG
   RUNG wire#w1
      Contact( #b_ERR_MON )
   END_RUNG wire#w2
   RUNG wire#w1
      Contact( #b_ERR_OP )
   END_RUNG wire#w2
   // the same network as SCL:
   IF #b_STARTING AND (NOT #IOP_COND OR #b_ERR_MON OR #b_ERR_OP) THEN #CMD_STEP := 1000; END_IF;
END_REGION

REGION Network 37: STEP MONITOR
   RUNG wire#powerrail
      Contact( #MON_EN )
      Contact( #b_STARTING )
      wire#w1
      { S7_Templates := "SrcType := Real" } LT_Contact(in1 := #r_MON, in2 := #MON_TIME)
      P_Contact(operand := #"Pulse 1HZ", bit := #PE_Mon)
      { S7_Templates := "SrcType := Real"; S7_GenerateENO := "TRUE" } Add(in1 := #r_MON, in2 := #SAMPLE_T, out => #r_MON)
   END_RUNG
   RUNG wire#w1
      Not()
      { S7_GenerateENO := "TRUE" } Move(in := 0.0, out1 => #r_MON)
   END_RUNG
   // the same network as SCL:
   #_w1 := #MON_EN AND #b_STARTING;
   #_w2 := #_w1 AND (#r_MON < #MON_TIME) AND #"Pulse 1HZ" AND NOT #PE_Mon;   // rising edge of #"Pulse 1HZ"
   #PE_Mon := #"Pulse 1HZ";
   IF #_w2 THEN #r_MON := #r_MON + #SAMPLE_T; END_IF;
   IF NOT #_w1 THEN #r_MON := 0.0; END_IF;
END_REGION

REGION Network 38: RESET IQRESET
END_REGION

REGION Network 39: RESET IQOPSTART
   RUNG wire#powerrail
      Contact( #IQOPSTART )
      R_Coil( #IQOPSTART )
   END_RUNG
   // the same network as SCL:
   IF #IQOPSTART THEN #IQOPSTART := FALSE; END_IF;
END_REGION

REGION Network 40: RESET IQOPHOLD
   RUNG wire#powerrail
      Contact( #IQOPHOLD )
      R_Coil( #IQOPHOLD )
   END_RUNG
   // the same network as SCL:
   IF #IQOPHOLD THEN #IQOPHOLD := FALSE; END_IF;
END_REGION

REGION Network 41: RESET IQOPSTOP
   RUNG wire#powerrail
      Contact( #IQOPSTOP )
      R_Coil( #IQOPSTOP )
   END_RUNG
   // the same network as SCL:
   IF #IQOPSTOP THEN #IQOPSTOP := FALSE; END_IF;
END_REGION

REGION Network 42: RESET IQOPCOMPLETE
   RUNG wire#powerrail
      Contact( #IQOPCOMPLETE )
      R_Coil( #IQOPCOMPLETE )
   END_RUNG
   // the same network as SCL:
   IF #IQOPCOMPLETE THEN #IQOPCOMPLETE := FALSE; END_IF;
END_REGION

REGION Network 43: DOSED QUANTITY
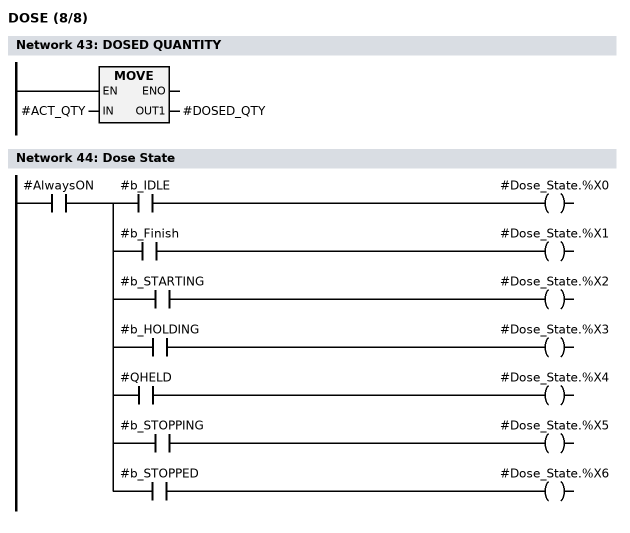
   RUNG wire#powerrail
      { S7_GenerateENO := "TRUE" } Move(in := #ACT_QTY, out1 => #DOSED_QTY)
   END_RUNG
   // the same network as SCL:
   #DOSED_QTY := #ACT_QTY;
END_REGION

REGION Network 44: Dose State
   RUNG wire#powerrail
      Contact( #AlwaysON )
      wire#w1
      Contact( #b_IDLE )
      Coil( #Dose_State.%X0 )
   END_RUNG
   RUNG wire#w1
      Contact( #b_Finish )
      Coil( #Dose_State.%X1 )
   END_RUNG
   RUNG wire#w1
      Contact( #b_STARTING )
      Coil( #Dose_State.%X2 )
   END_RUNG
   RUNG wire#w1
      Contact( #b_HOLDING )
      Coil( #Dose_State.%X3 )
   END_RUNG
   RUNG wire#w1
      Contact( #QHELD )
      Coil( #Dose_State.%X4 )
   END_RUNG
   RUNG wire#w1
      Contact( #b_STOPPING )
      Coil( #Dose_State.%X5 )
   END_RUNG
   RUNG wire#w1
      Contact( #b_STOPPED )
      Coil( #Dose_State.%X6 )
   END_RUNG
   // the same network as SCL:
   #Dose_State.%X0 := #AlwaysON AND #b_IDLE;
   #Dose_State.%X1 := #AlwaysON AND #b_Finish;
   #Dose_State.%X2 := #AlwaysON AND #b_STARTING;
   #Dose_State.%X3 := #AlwaysON AND #b_HOLDING;
   #Dose_State.%X4 := #AlwaysON AND #QHELD;
   #Dose_State.%X5 := #AlwaysON AND #b_STOPPING;
   #Dose_State.%X6 := #AlwaysON AND #b_STOPPED;
END_REGION
END_FUNCTION_BLOCK
